FUNCTION_BLOCK FB_SafetyCounter
VAR
	nSafetyCounterOC 	: UDINT;
	nSafetyCounterXMC1 	: UDINT;
	nSafetyCounterXMC2 	: UDINT;
	nSafetyCounterXMC3 	: UDINT;
	nSafetyCounterXMC4 	: UDINT;
	

	fbTimeoutOC : TON := (PT := PRG_ErrorHandling.tSafetyCounterTimeout);
	fbTimeoutXMC1 : TON := (PT := PRG_ErrorHandling.tSafetyCounterTimeout);
	fbTimeoutXMC2 : TON := (PT := PRG_ErrorHandling.tSafetyCounterTimeout);
	fbTimeoutXMC3 : TON := (PT := PRG_ErrorHandling.tSafetyCounterTimeout);
	fbTimeoutXMC4 : TON := (PT := PRG_ErrorHandling.tSafetyCounterTimeout);
	fbTimeoutEtherCAT : TON := (PT := PRG_ErrorHandling.tSafetyCounterTimeout);
	
	fbFrameCounter : FB_EcMasterFrameStatistic;
	bCount : BOOL;
	fFramesPerSecond : LREAL;
	
	bNoConnectionToOC : BOOL;
	bNoConnectionToXMC1 : BOOL;
	bNoConnectionToXMC2 : BOOL;
	bNoConnectionToXMC3 : BOOL;
	bNoConnectionToXMC4 : BOOL;
	bNoEtherCATConnection : BOOL;
END_VAR
VAR_INPUT
	bReset : BOOL;
END_VAR
VAR_OUTPUT
	nSafetyCounter : UDINT;
END_VAR

doEtherCATFrameCount();

nSafetyCounter := nSafetyCounter + 1;


//OC
IF PRG_MainController.stOperationControlCommands.nSafetyCounterOC <> nSafetyCounterOC THEN
	nSafetyCounterOC := PRG_MainController.stOperationControlCommands.nSafetyCounterOC;
	fbTimeoutOC(IN := FALSE);
	bNoConnectionToOC := FALSE;
ELSE
	fbTimeoutOC(IN := NOT bReset);
	bNoConnectionToOC := FALSE;
	IF fbTimeoutOC.Q THEN
		bNoConnectionToOC := TRUE;
	END_IF
END_IF

//XMC1
IF PRG_MainController.stXMCCommands.nSafetyCounterXMC1 <> nSafetyCounterXMC1 THEN
	nSafetyCounterXMC1 := PRG_MainController.stXMCCommands.nSafetyCounterXMC1;
	fbTimeoutXMC1(IN := FALSE);
	bNoConnectionToXMC1 := FALSE;
ELSE
	fbTimeoutXMC1(IN:= NOT bReset);
	bNoConnectionToXMC1 := FALSE;
	IF fbTimeoutXMC1.Q THEN
		bNoConnectionToXMC1 := TRUE;
	END_IF
END_IF

//XMC2
IF PRG_MainController.stXMCCommands.nSafetyCounterXMC2 <> nSafetyCounterXMC2 THEN
	nSafetyCounterXMC2 := PRG_MainController.stXMCCommands.nSafetyCounterXMC2;
	fbTimeoutXMC2(IN := FALSE);
	bNoConnectionToXMC2 := FALSE;
ELSE
	fbTimeoutXMC2(IN:= NOT bReset);
	bNoConnectionToXMC2 := FALSE;
	IF fbTimeoutXMC2.Q THEN
		bNoConnectionToXMC2 := TRUE;
	END_IF
END_IF

//XMC3
IF PRG_MainController.stXMCCommands.nSafetyCounterXMC3 <> nSafetyCounterXMC3 THEN
	nSafetyCounterXMC3 := PRG_MainController.stXMCCommands.nSafetyCounterXMC3;
	fbTimeoutXMC3(IN := FALSE);
	bNoConnectionToXMC3 := FALSE;
ELSE
	fbTimeoutXMC3(IN:= NOT bReset);
	bNoConnectionToXMC3 := FALSE;
	IF fbTimeoutXMC3.Q THEN
		bNoConnectionToXMC3 := TRUE;
	END_IF
END_IF

//XMC4
IF PRG_MainController.stXMCCommands.nSafetyCounterXMC4 <> nSafetyCounterXMC4 THEN
	nSafetyCounterXMC4 := PRG_MainController.stXMCCommands.nSafetyCounterXMC4;
	fbTimeoutXMC4(IN := FALSE);
	bNoConnectionToXMC4 := FALSE;
	fbTimeoutXMC1(IN := FALSE);
ELSE
	fbTimeoutXMC4(IN:= NOT bReset);
	bNoConnectionToXMC4 := FALSE;
	IF fbTimeoutXMC4.Q THEN
		bNoConnectionToXMC4 := TRUE;
	END_IF
END_IF

METHOD PRIVATE doEtherCATFrameCount
VAR_INPUT
END_VAR
IF NOT bCount THEN
	bCount := TRUE;
	fbFrameCounter(sNetId := '10.183.66.136.2.1', bExecute := bCount, fFramesPerSecond => fFramesPerSecond);
END_IF

IF bCount THEN
	bCount := FALSE;
	fbFrameCounter(sNetId := '10.183.66.136.2.1', bExecute := bCount, fFramesPerSecond => fFramesPerSecond);
END_IF

IF fFramesPerSecond <> 0 THEN
	bNoEtherCATConnection := FALSE;
	fbTimeoutEtherCAT(IN := FALSE);
ELSE
	fbTimeoutEtherCAT(IN := NOT bReset);
	bNoEtherCATConnection := FALSE;
	IF fbTimeoutEtherCAT.Q THEN
		bNoEtherCATConnection := TRUE;
	END_IF
END_IF
END_METHOD

PROPERTY PUBLIC nErrorID : UDINT
GET
nErrorID.0 := 	bNoConnectionToOC;
nErrorID.1 :=	bNoConnectionToXMC1;
nErrorID.2 :=	bNoConnectionToXMC2;
nErrorID.3 :=	bNoConnectionToXMC3;
nErrorID.4 := 	bNoConnectionToXMC4;
nErrorID.5 :=	bNoEtherCATConnection;
END_GET
END_PROPERTY

END_FUNCTION_BLOCK

(* stored: Version 1.1.0.1, ProductVersion 3.1.4024.12
   POU FB_SafetyCounter: Id {6f347c18-b88c-4382-a068-898d8214114a}, SpecialFunc None
   Method doEtherCATFrameCount: Id {4c37a95f-b91c-4db3-bee0-e47fcbc81cef}
   Property nErrorID: Id {eb85ba54-2be4-4713-9fe4-b6279706a220}
   Get Get: Id {4ce907e6-a3f0-49c3-adc0-5271cdbfc60e} *)
